# B&R Automation Studio project semesterprojektV005
Automation Studio 

## Logical view

### Global.var
```iecst
VAR
	dirX : BOOL;
	dirY : BOOL;
	dirZ : BOOL;
	enabX : BOOL;
	enabY : BOOL;
	enabZ : BOOL;
	drawFunction : BOOL;
	input : ARRAY[0..65000] OF USINT;
	posX : UDINT;
	posY : UDINT;
	posZ : UDINT;
	reset : BOOL;
	stepX : BOOL;
	stepY : BOOL;
	stepZ : BOOL;
	switch_X : BOOL;
	t : USINT;
	quit : BOOL;
	sharpen : UINT;
	status : USINT;
	testEnab : BOOL;
	z_move_down : BOOL;
	z_move_up : BOOL;
	y_move_right : BOOL;
	y_move_left : BOOL;
	x_move_right : BOOL;
	x_move_left : BOOL;
	sharpenderNeed : BOOL;
	switch_Z : BOOL;
	switch_Y : BOOL;
	percentage : REAL; (*%*)
	newLineX : UDINT;
	ValueZ : UINT;
	penLength : REAL;
	placeInArray : UDINT;
	placement : UINT;
	newLineHelper : UDINT;
END_VAR
```

### Program Logical/Draw

#### Variables.var
```iecst
VAR
	check : UDINT;
	sharpenderLen : UINT;
	timer : TON;
	i : UDINT;
	tempX : UDINT;
	activator : BOOL;
	finder : BOOL;
	tempPlace : UINT;
END_VAR
```

#### Main.st
```iecst
PROGRAM _INIT

	placeInArray := 0;
	i := 0;
	sharpen := 1;
	activator := FALSE;
	testEnab:= FALSE;
	penLength := 0;
	sharpenderNeed:= 0;

END_PROGRAM

PROGRAM _CYCLIC
	ValueZ := REAL_TO_INT(penLength**1.5);
	sharpenderLen := REAL_TO_INT(45000/penLength);

	IF (reset = FALSE AND testEnab = FALSE AND penLength > 5 ) THEN
//		percentage:= (UINT_TO_REAL(placeInString)/LEN(input))*100;

		IF switch_X = FALSE OR switch_Y = FALSE OR switch_Z = FALSE THEN
			enabX := TRUE;
			enabY := TRUE;
			enabZ := TRUE;
		END_IF

		IF (enabX = FALSE) THEN
			status:= 2;
		END_IF

		IF (i = 30) THEN
			IF placement = 20016 OR placement = 20017 THEN
				newLineHelper := newLineHelper - 17 ;
				posX := posX + 17;
			ELSIF placement = 21041 OR placement = 21040 THEN
				FOR check := placeInArray TO finder BY check +1 DO
					tempPlace := input[check];
					IF tempPlace = 21041 THEN
						finder := TRUE;
					ELSIF tempPlace = 20016 OR tempPlace = 20017 THEN
						placeInArray := check -1;
						newLineHelper := newLineHelper + 17;
						posX := posX - 17;
						finder := TRUE;
					END_IF
				END_FOR
			END_IF
			placeInArray := placeInArray + 1;
			i := 0;
		END_IF
		placement := input[placeInArray];

		// here the robot will move to the shapener, sharpen the pencil and move back to were it came from
		IF (sharpen >= 30000) THEN //!!!!!
			IF (posZ >= 300 AND tempX > 0 AND activator = FALSE) THEN  // !!!!!!
				dirZ := FALSE;
				stepZ := NOT stepZ;
				IF (stepZ = FALSE) THEN
					posZ := posZ -1;
				END_IF

			ELSIF (tempX > 0 AND posZ <= 300 AND activator = FALSE)THEN //!!!!!
				dirX := FALSE;
				stepX := NOT stepX;
				IF (stepX = FALSE) THEN
					tempX := tempX -1;
				END_IF

			ELSIF (tempX = 0 AND posZ <= 1500 + sharpenderLen AND activator = FALSE) THEN //!!!!!
				dirZ := TRUE;
				stepZ := NOT stepZ;
				IF (stepZ = FALSE) THEN
					posZ := posZ +1;
				END_IF

			ELSIF (tempX = 0 AND posZ >= 1500 + sharpenderLen AND activator = FALSE) THEN //!!!!!!
				timer.IN := TRUE;
				timer.PT := T#6000ms;
				IF timer.Q THEN
					activator := TRUE;
				END_IF

			ELSIF  (tempX = 0 AND posZ > 300 AND activator = TRUE) THEN//!!!!!
				dirZ := FALSE;
				stepZ := NOT stepZ;
				IF (stepZ = FALSE) THEN
					posZ := posZ - 1;
				END_IF

			ELSIF (tempX < posX  AND posZ = 300 AND activator = TRUE) THEN //!!!!!
				dirX := TRUE;
				stepX := NOT stepX;
				IF (stepX = FALSE) THEN
					tempX := tempX +1;
				END_IF

			ELSIF (tempX = posX  AND posZ = 300 AND activator = TRUE) THEN //!!!!!!
				sharpen := 0;
				activator := FALSE;
				timer.IN := FALSE;

			END_IF

		ELSE
			// here the robot will draw
			IF (placement = 21041 AND i < 30) THEN
				IF (posZ < (3200-ValueZ)) THEN  // !!!!!!
					IF dirZ THEN
						stepZ := NOT stepZ;
						IF (stepZ = FALSE) THEN
							posZ := posZ +1;
						END_IF
					ELSE
						dirZ := TRUE;
					END_IF

				ELSE
					IF dirX THEN
						stepX := NOT stepX;
						i := i + 1;
						IF (stepX = FALSE) THEN
							posX := posX + 1;
							newLineX := newLineX +1;
							sharpen := sharpen + 1;
							tempX := posX;
						END_IF
					ELSE
						dirX := TRUE;
					END_IF

				END_IF

			//dont draw
			ELSIF placement = 21040 AND i < 30 THEN
				IF (posZ > (2900-ValueZ)) THEN  // !!!!!!
					IF dirZ = FALSE THEN
						stepZ := NOT stepZ;
						IF (stepZ = FALSE) THEN
							posZ := posZ -1;
						END_IF
					ELSE
					dirZ := FALSE;
					END_IF
				ELSE
					IF dirX THEN
						stepX := NOT stepX;
						i := i + 1;
						IF (stepX = FALSE) THEN
							posX := posX +1;
							newLineX := newLineX +1;
						END_IF
					ELSE
						dirX := TRUE;
					END_IF

				END_IF

			ELSIF (placement = 20016 OR placement = 20017) THEN
				IF (posZ > (2900-ValueZ) )THEN  // !!!!!!
					IF dirZ = FALSE THEN
						stepZ := NOT stepZ;
						IF (stepZ = FALSE) THEN
							posZ := posZ -1;
						END_IF
					ELSE
						dirZ := FALSE;
					END_IF

				ELSIF (posZ <= (2900-ValueZ)) AND (newLineX >= (newLineHelper)) THEN//!!!!
					IF dirX = FALSE THEN
						stepX := NOT stepX;
						IF (stepX = FALSE) THEN
							posX := posX - 1;
							newLineX := newLineX -1;
						END_IF
					ELSE
						dirX := FALSE;
					END_IF

				ELSIF ((posZ <= (2900-ValueZ)) AND (newLineX <= newLineHelper) AND (i < 30)(* OR ( posZ = 0)*)) THEN
					IF dirY THEN
						stepY := NOT stepY;
						i := i +1;
						IF (stepY = FALSE) THEN
							posX := posX - 1;
							newLineX := newLineX -1;
						END_IF
					ELSE
						dirY := TRUE;
					END_IF

				END_IF

			ELSIF placement = 20785 OR placement = 20784 THEN

				quit := TRUE;
			END_IF

		END_IF

	END_IF
	timer();
END_PROGRAM

PROGRAM _EXIT

END_PROGRAM
```

### Program Logical/emergencyStop

#### Main.st
```iecst
PROGRAM _INIT
	// resets the values every time the PLC starts.
	reset_quit := FALSE;
	emergencyStop := FALSE;

END_PROGRAM

PROGRAM _CYCLIC
	IF (emergencyStop) THEN // emergency button
		enabX := TRUE;		// disables x-axis stepper
		enabY := TRUE;		// disables y-axis stepper
		enabZ := TRUE;		// disables Z-axis stepper
		status := 0;

	END_IF

	IF (reset_quit) THEN // Reset button
		reset := TRUE;		// starts the reset seqence in reset-program
		quit := TRUE;
		status := 1;		// sets status light to 1
		reset_quit := FALSE;
		placeInString := 0;	//resets place in array

	END_IF

END_PROGRAM

PROGRAM _EXIT
	(* Insert code here *)

END_PROGRAM
```

### Program Logical/reset

#### Variables.var
```iecst
VAR
	resetX : USINT;
	resetY : USINT;
	resetZ : USINT;
	timer : TON;
END_VAR
```

#### Main.st
```iecst
PROGRAM _INIT
	reset := TRUE;//
	resetX := 0;
	resetY := 0;
	resetZ := 0;

	quit := FALSE;
	status := 1;
	testEnab := TRUE;//
END_PROGRAM

PROGRAM _CYCLIC

//
	IF (reset = TRUE AND testEnab = FALSE) THEN
		IF switch_X = TRUE AND resetX = 0  THEN // Resets the x-axis
			enabX:= FALSE;
			dirX:= FALSE;

			stepX := NOT stepX;
		ELSIF switch_X = FALSE THEN
			resetX := 1;
			dirX:= TRUE;
			stepX := NOT stepX;
		END_IF

		IF switch_Y = TRUE AND resetY = 0 THEN // Resets the y-axis
			enabY:= FALSE;
			dirY:= FALSE;
			stepY := NOT stepY;
		ELSIF switch_Y = FALSE THEN
			resetY := 1;
			dirY:= TRUE;
			stepY := NOT stepY;
		END_IF

		IF switch_Z = TRUE AND resetZ = 0 THEN // Resets the z-axis
			enabZ:= FALSE;
			dirZ:= FALSE;
			stepZ := NOT stepZ;
		ELSIF switch_Z = FALSE THEN
			resetZ := 1;
			dirZ:= TRUE;
			stepZ := NOT stepZ;
		END_IF

// sets the position of the variables posX, posY and posZ
		timer.IN := TRUE;
		timer.PT := T#100ms;
		IF timer.Q THEN
			IF resetX = 1 AND resetY = 1 AND resetZ = 1 THEN
				posX := 0;
				posY := 0;
				posZ := 0;
				resetX := 2;
			END_IF
			timer.IN := FALSE;
		END_IF

	// if start-button pressed, then go to start position
		IF quit = FALSE AND resetX = 2 THEN
			IF posX < 1900 THEN
				dirX := TRUE;
				stepX := NOT stepX;
				IF (stepX = FALSE) THEN
					posX := posX +1;
				END_IF
			ELSE
				reset:= FALSE;
				resetX := 0;
				resetY := 0;
				resetZ := 0;
				newLineX :=  2294967295;
				newLineHelper := 2294967295;
			END_IF
		END_IF
	END_IF

	// move x-axis left
	IF (x_move_left AND testEnab) THEN
		stepX := NOT stepX;
		dirX := TRUE;
		IF stepX = FALSE THEN
			posX := posX +1;
		END_IF
	END_IF

	// move x-axis right
	IF (x_move_right AND testEnab) THEN
		stepX := NOT stepX;
		dirX := FALSE;
		IF stepX = FALSE THEN
			posX := posX -1;
		END_IF
	END_IF

	// move y-axis left
	IF (y_move_left AND testEnab) THEN
		stepY := NOT stepY;
		dirY := TRUE;
		IF stepY = FALSE THEN
			posY := posY +1;
		END_IF
	END_IF

	// move y-axis right
	IF (y_move_right AND testEnab) THEN
		stepY := NOT stepY;
		dirY := FALSE;
		IF stepY = FALSE THEN
			posY := posY -1;
		END_IF
	END_IF

	// move z-axis up
	IF (z_move_up AND testEnab) THEN
		stepZ := NOT stepZ;
		dirZ := FALSE;
		IF stepZ = FALSE THEN
			posZ := posZ -1;
		END_IF
	END_IF

	// move z-axis down
	IF (z_move_down AND testEnab) THEN
		stepZ := NOT stepZ;
		dirZ := TRUE;
		IF stepZ = FALSE THEN
			posZ := posZ +1;
		END_IF
	END_IF

	timer();
END_PROGRAM

PROGRAM _EXIT
	(* Insert code here *)

END_PROGRAM
```

### Program Logical/TCP

#### Variables.var
```iecst
VAR
	reciveData : ARRAY[0..199999] OF BOOL;
	tcp2 : TcpServer;
	tcp1 : TcpOpen;
	state : UINT;
	tcp3 : TcpRecv;
	tcp4 : TcpSend;
	tcp5 : TcpClose;
END_VAR
```

#### Main.st
```iecst
PROGRAM _INIT
	state := 1;

END_PROGRAM

PROGRAM _CYCLIC
	CASE state OF
		1:
			tcp1.enable := TRUE;
			tcp1.port := 12345;
			tcp1.options := tcpOPT_REUSEADDR;
			tcp1();
			IF tcp1.status = 0 THEN
				state := 10;
			END_IF

		10:
			tcp2.enable := TRUE;
			tcp2.ident := tcp1.ident;
			tcp2();
			IF tcp2.status = 0 THEN
				state := 20;
			END_IF

		20:
			tcp3.enable := TRUE;
			tcp3.ident := tcp2.identclnt;
			tcp3.pData := ADR(input);
			tcp3.datamax := SIZEOF (input);
			tcp3();
			IF tcp3.status = 0 THEN
				//input := reciveData;
				//				FOR i := 0 TO i = 2000 BY i + 1 DO
				//					test.IN := reciveData[i];
				//					input := CONCAT(input, test.Q);
				//				END_FOR
				state := 30;

			END_IF

		30:
			tcp4.enable := TRUE;
			tcp4.ident := tcp2.identclnt;
			tcp4.pData := ADR(input);
			tcp4.datalen := brsstrlen(ADR(input));
			tcp4();
			IF tcp4.status = 0 THEN
				state := 40;
			END_IF

		40:
			tcp5.enable := TRUE;
			tcp5.ident := tcp2.identclnt;
			tcp5();
			IF tcp5.status = 0 THEN
				tcp2.enable := FALSE;
				state := 10;

				//				FOR i := 0 TO i < 200 BY i + 1 DO
				//					reciveData[i] := 0;
				//				END_FOR
			END_IF
	END_CASE
//	test();
END_PROGRAM

PROGRAM _EXIT
	tcp5.enable := TRUE;
	tcp5.ident := tcp2.identclnt;
	tcp5();

	tcp5.enable := TRUE;
	tcp5.ident := tcp1.ident;
	tcp5();

END_PROGRAM
```
